// TIA Portal V20 export
VAR_GLOBAL   // PLC tag table "SR-X100W_Exit"
   Exit_Read_Complete AT %I858.0 : Bool;
   Exit_Read_Failure AT %I859.0 : Bool;
   Exit_Read_Data AT %I860.0 : "SR-X100W_Read_Data";
   Exit_Read_Request AT %Q858.0 : Bool;
   Exit_Read_Complete_Clear AT %Q859.0 : Bool;
END_VAR
